(* IEC 61131-3 sources: Industry-PLC-LLM/data/PLCBEAD_repo/PLCBEAD_PLCEmbed-main/PLC-BEAD/Source/GEB/MINUTE, 1 file *)

(* ---- MINUTE.ST ---- *)
FUNCTION MINUTE:INT

	VAR_INPUT
		ITOD :	UDINT;
	END_VAR

	minute := UDINT_TO_INT((itod / UDINT#60000) - ((itod / UDINT#3600000) * UDINT#60));

END_FUNCTION

PROGRAM program0
  VAR
	  ITOD :	UDINT;
    CEIL5_OUT : INT;
  END_VAR

  CEIL5_OUT := MINUTE(ITOD);
END_PROGRAM
